// TIA Portal project "P2" (V17)

(* hardware
DEVICE "S7-1500/ET200MP station_1"  S7-1500 station
   slot 0: "Rail_0"  Rack  6ES7 590-1***0-0AA0
   slot 1: "PLC_1"  CPU 1515-2 PN  6ES7 515-2AM02-0AB0  V2.9
      slot 3: "CPU display_1"  6ES7591-1BA00-0AA0
      slot 32768: "PROFINET interface_1"  X1
         slot 32769: "Port_1"  X1 P1
         slot 32770: "Port_2"  X1 P2
      slot 33024: "PROFINET interface_2"  X2
         slot 33025: "Port_1"  X2 P1
      slot 34817: "Virtual CP interface port_1"  Virtual CP interface port  Virtual CP interface port
*)

// ===== PLC "PLC_1"  CPU 1515-2 PN =====

VAR_GLOBAL   // PLC tag table "Default tag table"
   "System ON" AT %E0.0 : Bool;   // ENCENDIDO
   "S1" AT %E0.1 : Bool;   // SENSOR (I/O) PLANTA BAJA
   "P1" AT %M0.0 : Bool;
   "GREEN LIGHT PLANTA BAJA" AT %A0.0 : Bool;   // GREEN LIGHT (I/O) PLANTA BAJA
   "GREEN LIGHT SOTANO" AT %A0.1 : Bool;   // GREEN LIGHT (I/O) SOTANO
   "RED LIGHT PLANTA BAJA" AT %A0.2 : Bool;   // RED LIGHT (I/O) PLANTA BAJA
   "RED LIGHT SOTANO" AT %A0.3 : Bool;   // RED LIGHT (I/O) SOTANO
   "P2" AT %M0.1 : Bool;
   "CAR PASS S1" AT %M10.0 : Bool;   // EL CARRO PASA EL SENSOR 1
   "CAR PASS S2" AT %M10.3 : Bool;   // EL CARRO PASA EL SENSOR 2
   "S2" AT %E0.2 : Bool;
   "P3" AT %M0.3 : Bool;
   "TAG_8" AT %M11.0 : Bool;
   "TAG_9" AT %M11.1 : Bool;
   "TAG_12" AT %M11.2 : Bool;
   "TAG_13" AT %M11.3 : Bool;
   "TAG_5" AT %MB0 : Byte;
   "TAG_6" AT %AB0 : Byte;
   "TAG_7" AT %MB10 : Byte;
END_VAR

ORGANIZATION_BLOCK "Main"   // OB1, LAD, ProgramCycle
TITLE = "Main Program Sweep (Cycle)"
{ S7_Optimized_Access := 'TRUE' }
VERSION : 0.1
   VAR_INPUT
      Initial_Call : Bool;   // Initial call of this OB
      Remanence : Bool;   // =True, if remanent data are available
   END_VAR
   VAR_TEMP
      Tag_8 : Bool;
      Tag_9 : Bool;
   END_VAR
   VAR_TEMP   // added for the SCL form of the ladder/FBD networks
      _w1 : Bool;
      _w2 : Bool;
      _w3 : Bool;
      _w4 : Bool;
   END_VAR
BEGIN

REGION Network 1: GREEN LIGHT ENCENDIDO CUANDO EL SISTEMA ESTA ENCENDIDO - Primer Ciclo de escaneo
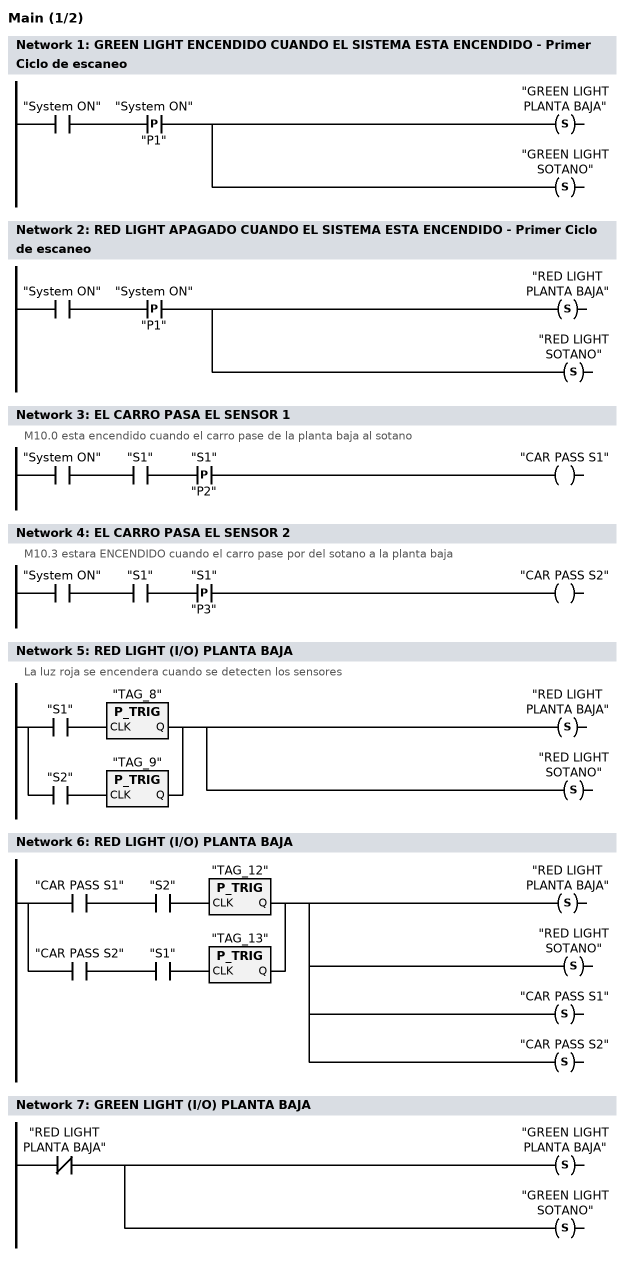
   RUNG wire#powerrail
      Contact( "System ON" )
      P_Contact(operand := "System ON", bit := "P1")
      wire#w1
      S_Coil( "GREEN LIGHT PLANTA BAJA" )
   END_RUNG
   RUNG wire#w1
      S_Coil( "GREEN LIGHT SOTANO" )
   END_RUNG
   // the same network as SCL:
   #_w1 := "System ON" AND "System ON" AND NOT "P1";   // rising edge of "System ON"
   "P1" := "System ON";
   IF #_w1 THEN
       "GREEN LIGHT PLANTA BAJA" := TRUE;
       "GREEN LIGHT SOTANO" := TRUE;
   END_IF;
END_REGION

REGION Network 2: RED LIGHT APAGADO CUANDO EL SISTEMA ESTA ENCENDIDO - Primer Ciclo de escaneo
   RUNG wire#powerrail
      Contact( "System ON" )
      P_Contact(operand := "System ON", bit := "P1")
      wire#w1
      S_Coil( "RED LIGHT PLANTA BAJA" )
   END_RUNG
   RUNG wire#w1
      S_Coil( "RED LIGHT SOTANO" )
   END_RUNG
   // the same network as SCL:
   #_w1 := "System ON" AND "System ON" AND NOT "P1";   // rising edge of "System ON"
   "P1" := "System ON";
   IF #_w1 THEN
       "RED LIGHT PLANTA BAJA" := TRUE;
       "RED LIGHT SOTANO" := TRUE;
   END_IF;
END_REGION

REGION Network 3: EL CARRO PASA EL SENSOR 1
   // M10.0 esta encendido cuando el carro pase de la planta baja al sotano
   RUNG wire#powerrail
      Contact( "System ON" )
      Contact( "S1" )
      P_Contact(operand := "S1", bit := "P2")
      Coil( "CAR PASS S1" )
   END_RUNG
   // the same network as SCL:
   #_w1 := "System ON" AND "S1" AND "S1" AND NOT "P2";   // rising edge of "S1"
   "P2" := "S1";
   "CAR PASS S1" := #_w1;
END_REGION

REGION Network 4: EL CARRO PASA EL SENSOR 2
   // M10.3 estara ENCENDIDO cuando el carro pase por del sotano a la planta baja
   RUNG wire#powerrail
      Contact( "System ON" )
      Contact( "S1" )
      P_Contact(operand := "S1", bit := "P3")
      Coil( "CAR PASS S2" )
   END_RUNG
   // the same network as SCL:
   #_w1 := "System ON" AND "S1" AND "S1" AND NOT "P3";   // rising edge of "S1"
   "P3" := "S1";
   "CAR PASS S2" := #_w1;
END_REGION

REGION Network 5: RED LIGHT (I/O) PLANTA BAJA
   // La luz roja se encendera cuando se detecten los sensores
   RUNG wire#powerrail
      Contact( "S1" )
      P_Trig( "TAG_8" )
      wire#w1
      S_Coil( "RED LIGHT PLANTA BAJA" )
   END_RUNG
   RUNG wire#powerrail
      Contact( "S2" )
      P_Trig( "TAG_9" )
   END_RUNG wire#w1
   RUNG wire#w1
      S_Coil( "RED LIGHT SOTANO" )
   END_RUNG
   // the same network as SCL:
   #_w1 := "S1" AND NOT "TAG_8";   // rising edge
   "TAG_8" := "S1";
   #_w2 := "S2" AND NOT "TAG_9";   // rising edge
   "TAG_9" := "S2";
   IF #_w1 OR #_w2 THEN
       "RED LIGHT PLANTA BAJA" := TRUE;
       "RED LIGHT SOTANO" := TRUE;
   END_IF;
END_REGION

REGION Network 6: RED LIGHT (I/O) PLANTA BAJA
   RUNG wire#powerrail
      Contact( "CAR PASS S1" )
      Contact( "S2" )
      P_Trig( "TAG_12" )
      wire#w1
      S_Coil( "RED LIGHT PLANTA BAJA" )
   END_RUNG
   RUNG wire#powerrail
      Contact( "CAR PASS S2" )
      Contact( "S1" )
      P_Trig( "TAG_13" )
   END_RUNG wire#w1
   RUNG wire#w1
      S_Coil( "RED LIGHT SOTANO" )
   END_RUNG
   RUNG wire#w1
      S_Coil( "CAR PASS S1" )
   END_RUNG
   RUNG wire#w1
      S_Coil( "CAR PASS S2" )
   END_RUNG
   // the same network as SCL:
   #_w1 := "CAR PASS S1" AND "S2";
   #_w2 := #_w1 AND NOT "TAG_12";   // rising edge
   "TAG_12" := #_w1;
   #_w3 := "CAR PASS S2" AND "S1";
   #_w4 := #_w3 AND NOT "TAG_13";   // rising edge
   "TAG_13" := #_w3;
   IF #_w2 OR #_w4 THEN
       "RED LIGHT PLANTA BAJA" := TRUE;
       "RED LIGHT SOTANO" := TRUE;
       "CAR PASS S1" := TRUE;
       "CAR PASS S2" := TRUE;
   END_IF;
END_REGION

REGION Network 7: GREEN LIGHT (I/O) PLANTA BAJA
   RUNG wire#powerrail
      I_Contact( "RED LIGHT PLANTA BAJA" )
      wire#w1
      S_Coil( "GREEN LIGHT PLANTA BAJA" )
   END_RUNG
   RUNG wire#w1
      S_Coil( "GREEN LIGHT SOTANO" )
   END_RUNG
   // the same network as SCL:
   IF NOT "RED LIGHT PLANTA BAJA" THEN
       "GREEN LIGHT PLANTA BAJA" := TRUE;
       "GREEN LIGHT SOTANO" := TRUE;
   END_IF;
END_REGION

REGION Network 8: GREEN LIGHT (I/O) PLANTA BAJA
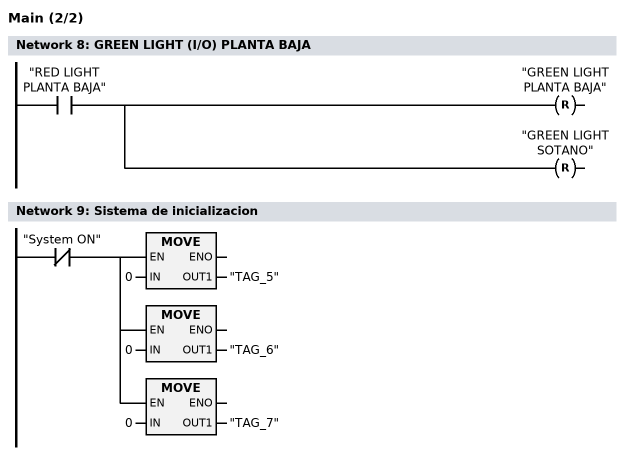
   RUNG wire#powerrail
      Contact( "RED LIGHT PLANTA BAJA" )
      wire#w1
      R_Coil( "GREEN LIGHT PLANTA BAJA" )
   END_RUNG
   RUNG wire#w1
      R_Coil( "GREEN LIGHT SOTANO" )
   END_RUNG
   // the same network as SCL:
   IF "RED LIGHT PLANTA BAJA" THEN
       "GREEN LIGHT PLANTA BAJA" := FALSE;
       "GREEN LIGHT SOTANO" := FALSE;
   END_IF;
END_REGION

REGION Network 9: Sistema de inicializacion
   RUNG wire#powerrail
      I_Contact( "System ON" )
      wire#w1
      Move(in := 0, out1 => "TAG_5")
   END_RUNG
   RUNG wire#w1
      Move(in := 0, out1 => "TAG_6")
   END_RUNG
   RUNG wire#w1
      Move(in := 0, out1 => "TAG_7")
   END_RUNG
   // the same network as SCL:
   IF NOT "System ON" THEN
       "TAG_5" := 0;
       "TAG_6" := 0;
       "TAG_7" := 0;
   END_IF;
END_REGION
END_ORGANIZATION_BLOCK